// TwinCAT 3 PLC project MotorProject
// ProgramVersion: 3.1.4023.0
// libraries:
//   Tc2_MC2, * (Beckhoff Automation GmbH)
//   Tc2_Standard, * (Beckhoff Automation GmbH)
//   Tc2_System, * (Beckhoff Automation GmbH)
//   Tc3_Module, * (Beckhoff Automation GmbH)
// project tree:
//   DUTs/ tDriveOutNCtrl1.TcDUT (not stored), tEncOutNCtrl1.TcDUT (not stored), tDriveInNState1.TcDUT (not stored), tDriveInNState2.TcDUT (not stored), tEncInState1.TcDUT, tEncInState2.TcDUT
//   GVLs/ IO.TcGVL
//   / PlcTask.TcTTO (not stored)
//   POUs/ MAIN.TcPOU, Motor.TcPOU (not stored)
// real-time tasks:
//   TASK PlcTask: cycle T#10ms, priority 20, ADS port 350
// motion (NC):
//   TASK NC-Task 1 SAF: cycle T#2ms, priority 4, ADS port 501
//   TASK NC-Task 1 SVB: cycle T#10ms, priority 8, ADS port 511
//   AXIS Axis 1 (id 1)
//     Dynamic: Acceleration=750, Deceleration=750, Jerk=1125
//     Velo: Maximum=1000
//     OtherSettings: AllowMotionCmdToSlave=true
//     encoder EncType=4
//       EncPara: MaxCount=#x0000ffff
//         Inc: RefSoftSyncMask=#x0000ffff
//     drive DrvType=23
//       Analog: TorqueSetpointScale=10, ScaleFactorActTorque=0.1
//       TimeComp: TaskDelayCycles=1
//     controller CtrType=1
//       CtrPara: PriorControlFactor=1
//         PosDiffControl: Enable=false
//         Observer: BandWidth=20
//   AXIS Axis 2 (id 2)
//     OtherSettings: AllowMotionCmdToSlave=true
//     encoder EncType=4
//       EncPara: MaxCount=#x0000ffff
//         Inc: RefSoftSyncMask=#x0000ffff
//     drive DrvType=23
//       Analog: TorqueSetpointScale=10, ScaleFactorActTorque=0.1
//       TimeComp: TaskDelayCycles=1
//     controller CtrType=1
//       CtrPara: PriorControlFactor=1
//         Observer: BandWidth=20
//   AXIS Achse 3 (id 3)
//     OtherSettings: AllowMotionCmdToSlave=true
//     encoder EncType=4
//       EncPara: MaxCount=#x0000ffff
//         Inc: RefSoftSyncMask=#x0000ffff
//     drive DrvType=23
//       Analog: TorqueSetpointScale=10, ScaleFactorActTorque=0.1
//       TimeComp: TaskDelayCycles=1
//     controller CtrType=1
//       CtrPara: PriorControlFactor=1
//         Observer: BandWidth=20
//   AXIS Achse 4 (id 4)
//     OtherSettings: AllowMotionCmdToSlave=true
//     encoder EncType=1
//       Inc: RefSoftSyncMask=#x0000ffff
//     drive DrvType=5
//       Analog: TorqueSetpointScale=10, ScaleFactorActTorque=0.1
//       TimeComp: TaskDelayCycles=1
//     controller CtrType=1
//       CtrPara: PriorControlFactor=1
//         Observer: BandWidth=20
//   AXIS Achse 5 (id 5)
//     OtherSettings: AllowMotionCmdToSlave=true
//     encoder EncType=1
//     drive DrvType=5
//       Analog: TorqueSetpointScale=10, ScaleFactorActTorque=0.1
//       TimeComp: TaskDelayCycles=1
//     controller CtrType=1
//       CtrPara: PriorControlFactor=1
//         Observer: BandWidth=20
// variable links:
//   MotorProject/MotorProject Instance <-> NC-Task 1 SAF/Axes/Axis 1
//     PlcTask Inputs/MAIN.DriveOutNCtrl1/Enable <-> Drive/Outputs/Out/nCtrl1
//     PlcTask Inputs/MAIN.DriveOutNCtrl1/ReduceTorque <-> Drive/Outputs/Out/nCtrl1 @bit 2
//     PlcTask Inputs/MAIN.DriveOutNCtrl1/Reset <-> Drive/Outputs/Out/nCtrl1 @bit 1
//     PlcTask Inputs/MAIN.DriveOutNCtrl1/ThresholdActive <-> Drive/Outputs/Out/nCtrl1 @bit 3
//     PlcTask Inputs/MAIN.DriveOutNDataOut2 <-> Drive/Outputs/Out/nDataOut2[0]
//     PlcTask Inputs/MAIN.EncOutNCtrl1/EnableLatchExternNegativeEdge <-> Enc/Outputs/Out/nCtrl1 @bit 2
//     PlcTask Inputs/MAIN.EncOutNCtrl1/EnableLatchExternPositiveEdge <-> Enc/Outputs/Out/nCtrl1
//     PlcTask Inputs/MAIN.EncOutNCtrl1/SetCounter <-> Enc/Outputs/Out/nCtrl1 @bit 1
//     PlcTask Inputs/MAIN.EncOutNDataOut1 <-> Enc/Outputs/Out/nDataOut1[0]
//     PlcTask Outputs/MAIN.EncInData1 <-> Enc/Inputs/In/nDataIn1[0]
//     PlcTask Outputs/MAIN.EncInData2 <-> Enc/Inputs/In/nDataIn2[0]
//     PlcTask Outputs/MAIN.EncInState1/CounterOverflow <-> Enc/Inputs/In/nState1 @bit 3
//     PlcTask Outputs/MAIN.EncInState1/CounterUnderflow <-> Enc/Inputs/In/nState1 @bit 2
//     PlcTask Outputs/MAIN.EncInState1/ExtrpolationStall <-> Enc/Inputs/In/nState1 @bit 4
//     PlcTask Outputs/MAIN.EncInState1/LatchExternValid <-> Enc/Inputs/In/nState1
//     PlcTask Outputs/MAIN.EncInState1/SetCounterDone <-> Enc/Inputs/In/nState1 @bit 1
//     PlcTask Outputs/MAIN.EncInState2/StatusExternLatch <-> Enc/Inputs/In/nState2 @bit 2
//     PlcTask Outputs/MAIN.EncInState2/StatusInputA <-> Enc/Inputs/In/nState2
//     PlcTask Outputs/MAIN.EncInState2/StatusInputB <-> Enc/Inputs/In/nState2 @bit 1
//     PlcTask Outputs/MAIN.EncInState2/SyncError <-> Enc/Inputs/In/nState2 @bit 3
//     PlcTask Outputs/MAIN.EncInState2/TxPdoToggle <-> Enc/Inputs/In/nState2 @bit 4
//     PlcTask Outputs/MAIN.driveInState1/Error <-> Drive/Inputs/In/nState1 @bit 3
//     PlcTask Outputs/MAIN.driveInState1/MovingNegative <-> Drive/Inputs/In/nState1 @bit 5
//     PlcTask Outputs/MAIN.driveInState1/MovingPositive <-> Drive/Inputs/In/nState1 @bit 4
//     PlcTask Outputs/MAIN.driveInState1/Ready <-> Drive/Inputs/In/nState1 @bit 1
//     PlcTask Outputs/MAIN.driveInState1/ReadyToEnable <-> Drive/Inputs/In/nState1
//     PlcTask Outputs/MAIN.driveInState1/TorqueReduced <-> Drive/Inputs/In/nState1 @bit 6
//     PlcTask Outputs/MAIN.driveInState1/Warning <-> Drive/Inputs/In/nState1 @bit 2
//     PlcTask Outputs/MAIN.driveInState2/DigitalInput1 <-> Drive/Inputs/In/nState2
//     PlcTask Outputs/MAIN.driveInState2/DigitalInput2 <-> Drive/Inputs/In/nState2 @bit 1
//     PlcTask Outputs/MAIN.driveInState2/SyncError <-> Drive/Inputs/In/nState2 @bit 2
//     PlcTask Outputs/MAIN.driveInState2/TcPdoToggle <-> Drive/Inputs/In/nState2 @bit 3

// ---- DUTs/tEncInState1.TcDUT
TYPE tEncInState1 :
STRUCT
	LatchExternValid		: BIT;
	SetCounterDone			: BIT;
	CounterUnderflow		: BIT;
	CounterOverflow			: BIT;
	ExtrpolationStall		: BIT;
END_STRUCT
END_TYPE

// ---- DUTs/tEncInState2.TcDUT
TYPE tEncInState2 :
STRUCT	
	StatusInputA			: BIT;
	StatusInputB			: BIT;
	StatusExternLatch		: BIT;
	SyncError				: BIT;
	TxPdoToggle				: BIT;
END_STRUCT
END_TYPE

// ---- GVLs/IO.TcGVL
{attribute 'qualified_only'}
VAR_GLOBAL
	bOut1 	AT%Q*	: BOOL;
	bIn1 	AT%I*	: BOOL;	
END_VAR

// ---- POUs/MAIN.TcPOU
PROGRAM MAIN
VAR
	
driveInState1 	AT%Q* 	: tDriveInNState1;
driveInState2 	AT%Q* 	: tDriveInNState2;
EncInState1		AT%Q*	: tEncInState1;
EncInState2		AT%Q*	: tEncInState2;
EncInData1		AT%Q*	: UINT;			// CounterValue
EncInData2		AT%Q*	: UINT;			// LatchValue

EncOutNCtrl1	AT%I*	: tEncOutNCtrl1;			// LatchValue
EncOutNDataOut1	AT%I*	: UINT;			// SetCounterValue

DriveOutNCtrl1	AT%I*	: tDriveOutNCtrl1;
DriveOutNDataOut2	AT%I*	: INT;		// Velocity

test : MDP5001_511_733_FFF278FE;

motor : Motor;


END_VAR



// motor(velocity:= DriveOutNDataOut2, counter=> EncInData1);

END_PROGRAM
